{attribute 'qualified_only'}
{attribute 'strict'}
{attribute 'to_string'}
TYPE E_3102_Position_initialize_status : (
		Failed	  := 0,
		Succeeded := 1
	) UINT;
END_TYPE

(* stored: Version 1.1.0.1, ProductVersion 3.1.4026.17
   DUT E_3102_Position_initialize_status: Id {172ee80c-2549-47bb-94ff-b2cefce7b056} *)
